// TIA Portal V17 export
FUNCTION "串联后分叉" : Void   // FC, LAD
{ S7_Optimized_Access := 'TRUE' }
VERSION : 0.1
// stored: AutoNumber true, IsIECCheckEnabled false, SetENOAutomatically false
BEGIN

REGION Network 1
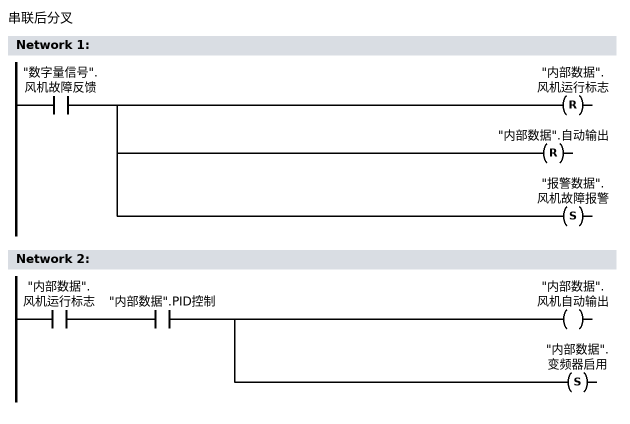
   RUNG wire#powerrail
      Contact( "数字量信号".风机故障反馈 )
      wire#w1
      R_Coil( "内部数据".风机运行标志 )
   END_RUNG
   RUNG wire#w1
      R_Coil( "内部数据".自动输出 )
   END_RUNG
   RUNG wire#w1
      S_Coil( "报警数据".风机故障报警 )
   END_RUNG
   // the same network as SCL:
   IF "数字量信号".风机故障反馈 THEN
       "内部数据".风机运行标志 := FALSE;
       "内部数据".自动输出 := FALSE;
       "报警数据".风机故障报警 := TRUE;
   END_IF;
END_REGION

REGION Network 2
   RUNG wire#powerrail
      Contact( "内部数据".风机运行标志 )
      Contact( "内部数据".PID控制 )
      wire#w1
      Coil( "内部数据".风机自动输出 )
   END_RUNG
   RUNG wire#w1
      S_Coil( "内部数据".变频器启用 )
   END_RUNG
   // the same network as SCL:
   "内部数据".风机自动输出 := "内部数据".风机运行标志 AND "内部数据".PID控制;
   IF "内部数据".风机自动输出 THEN "内部数据".变频器启用 := TRUE; END_IF;
END_REGION
END_FUNCTION
